// TIA Portal V20 export
// export: Created 2025-12-01T14:56:17.6771798Z, ExportSetting None, DisplayName Totally Integrated Automation Portal, DisplayVersion V20 Update 3, DisplayName TIA Portal Openness, DisplayVersion V20 Update 3, DisplayName TIA Portal Version Control Interface, DisplayVersion V20 Update 3, DisplayName STEP 7 Professional, DisplayVersion V20 Update 3, DisplayName STEP 7 Safety, DisplayVersion V20 Update 2, DisplayName WinCC Basic/Comfort/Advanced, DisplayVersion V20 Update 3, DisplayName WinCC Professional, DisplayVersion V20 Update 3, DisplayName WinCC Unified, DisplayVersion V20 Update 3
TYPE "UDT_ScadaEntradasZona"
   STRUCT
      Bit_00 : Bool;
      Marcha : Bool;   // Pulsador de Marcha
      Rearme : Bool;   // Pulsador de Rearme
      TestLuces : Bool;   // Pulsador de Test de Luces
      Auto : Bool;   // Selector de Automatico
      Paro : Bool;   // Pulsador de Paro
      Bit_06 : Bool;
      Bit_07 : Bool;
      Off_Line : Bool;
      Maintenimiento : Bool;
      Bit_12 : Bool;
      Bit_13 : Bool;
      Bit_14 : Bool;
      Bit_15 : Bool;
      Bit_16 : Bool;
      Bit_17 : Bool;
   END_STRUCT;
END_TYPE
